RoboDK station: MiniProject.rdk

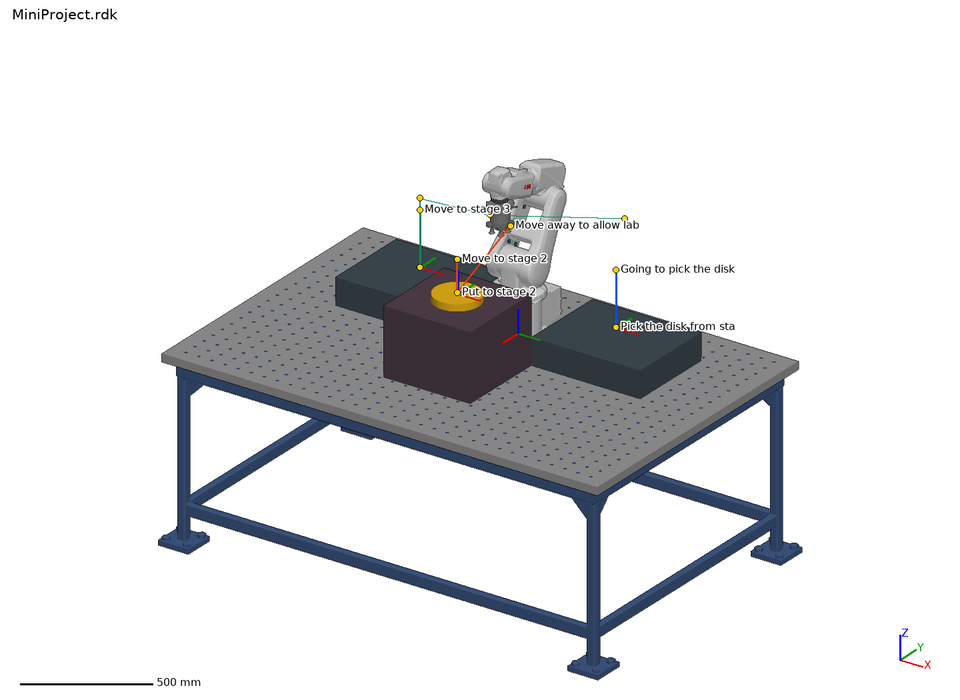
[picture v0: the station drawn from its stored meshes, robots at their saved joint values, targets as dots, program paths as lines]
Station MiniProject (saved by RoboDK 5.6.1). Poses are relative to the parent item; angles as X-Y-Z fixed-axis rotations.
  - object Table 2000x1200x800mm at (-630, -250, 0) mm, size 2020 x 1340 x 800 mm, geometry from Table-2000x1200x800mm.sld
  - object Stage 1 at (200, -200, 0) mm, size 500 x 400 x 120 mm, geometry from LINEW=0.500
  - object Stage 2 at (-200, -600, 0) mm, size 400 x 400 x 300 mm, geometry from LINEW=0.500
  - object Stage 2 at (-700, -200, 0) mm, size 500 x 400 x 120 mm, geometry from LINEW=0.500
  - frame ABB IRB 1100-4/0.58 Base at (0, 0, 0) mm, rotated rx 0 ry 0 rz -90 deg
    - robot ABB IRB 120-3/0.6: 6 axes, payload 3 kg, reach 580 mm, repeatability 0.01 mm, weight 25 kg
        modified DH rows (alpha deg, a mm, theta deg, d mm): 0, 0, 0, 290; -90, 0, -90, 0; 0, 270, 0, 0; -90, 70, 0, 302; 90, 0, 0, 0; -90, 0, 180, 72
        joint limits [-165, -110, -90, -160, -120, -400] to [165, 110, 70, 160, 120, 400]; home [0, 0, 0, 0, 0, 0]; saved at [0, -33.333, 16.582, 0, 106.741, 0]
      - tool SMC ZXP7A01-ZP20U-X1 Vacuum Gripper, TCP at (0, 0, 125) mm, size 88 x 106.8 x 127.9 mm
  - frame Frame 1 at (450, 0, 150) mm
    - target Going to pick the disk (Cartesian target) at (0, 0, 240) mm, rotated rx 180 ry 0 rz -180 deg; joints [0, 32.452, -33.546, 0, 91.094, 0] of ABB IRB 120-3/0.6
    - target Pick the disk from stage 1 (Cartesian target) at (0, 0, 0) mm, rotated rx 180 ry 0 rz -180 deg; joints [0, 47.712, -9.811, 0, 52.099, 0] of ABB IRB 120-3/0.6
  - frame Frame 2 at (0, -390, 320) mm
    - target Move to stage 2 (Cartesian target) at (0, -10, 150) mm, rotated rx 180 ry 0.01 rz 90 deg; joints [-90, 22.932, -35.32, 0, 102.378, 0] of ABB IRB 120-3/0.6
    - target Put to stage 2 (Cartesian target) at (0, -10, 10) mm, rotated rx 180 ry 0.01 rz 90 deg; joints [-90, 22.53, -7.796, 0, 75.256, 0] of ABB IRB 120-3/0.6
    - target Move away to allow label (Cartesian target) at (0, 340.58, 149.94) mm, rotated rx 180 ry 0.01 rz 90 deg; joints [-90, -49.057, 21.325, 0, 117.722, 0] of ABB IRB 120-3/0.6
    - target Pickup Again from stage 2 (Cartesian target) at (0, -10, 10) mm, rotated rx 180 ry 0.01 rz 90 deg; joints [-90, 22.53, -7.796, 0, 75.256, 0] of ABB IRB 120-3/0.6
    - target Move to up again from stage 2 (Cartesian target) at (0, -10, 150) mm, rotated rx 180 ry 0.01 rz 90 deg; joints [-90, 22.932, -35.32, 0, 102.378, 0] of ABB IRB 120-3/0.6
    - object Disk at (0, -10.01, -20) mm, rotated rx 0 ry -0.01 rz -90 deg, size 200 x 200 x 30 mm, geometry from LINEW=0.500
  - frame Frame 3 at (-450, 0, 150) mm
    - target Move to stage 3 (Cartesian target) at (0, 0, 240) mm, rotated rx -180 ry 0 rz -180 deg; joints [-180, 32.452, -33.546, 0, 91.094, 180] of ABB IRB 120-3/0.6
    - target Put on stage 2 (Cartesian target) at (0, 0, 0) mm, rotated rx -180 ry 0 rz -180 deg; joints [-180, 47.712, -9.811, 0, 52.099, 180] of ABB IRB 120-3/0.6
    - target End point 1 (Cartesian target) at (0, 0, 290) mm, rotated rx -180 ry 0 rz -180 deg; joints [-180, 34.445, -46.237, 0, 101.791, 180] of ABB IRB 120-3/0.6
    - target End Point 2 (Cartesian target) at (320, 0, 310) mm, rotated rx -180 ry 0 rz -180 deg; joints [-180, -33.964, 18.471, 0, 105.493, 180] of ABB IRB 120-3/0.6
    - target End point 3 (Cartesian target) at (939, 0, 467) mm, rotated rx 0 ry 90 rz 0 deg; joints [0, 0, 0, 0, 0, 0] of ABB IRB 120-3/0.6
  - program Replace disk 1 (1 instructions, listed below)
  - program Pick 1 (6 instructions, listed below)
  - program Place part 1 (9 instructions, listed below)
  - program Place part 2 (9 instructions, listed below)
  - program MainProgram (4 instructions, listed below)
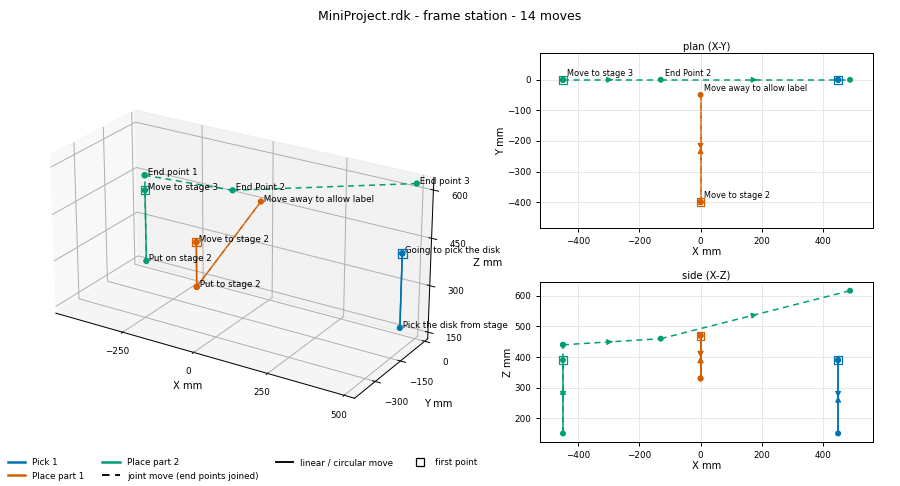
[picture p0: tool path of MiniProject.rdk in frame station, 14 of 14 moves have a stored position in this frame; points joined in program order, loops and branches not executed]

--- program Replace disk 1 (robot ABB IRB 120-3/0.6) ---
  Replace objects

--- program Pick 1 (robot ABB IRB 120-3/0.6) ---
  Set Ref.: Frame 1
  Set Tool: SMC ZXP7A01-ZP20U-X1 Vacuum Gripper
  MoveJ (Going to pick the disk)
  MoveL (Pick the disk from stage 1)
  Attach to SMC ZXP7A01-ZP20U-X1 Vacuum Gripper
  MoveL (Going to pick the disk)

--- program Place part 1 (robot ABB IRB 120-3/0.6) ---
  Set Ref.: Frame 2
  Set Tool: SMC ZXP7A01-ZP20U-X1 Vacuum Gripper
  MoveJ (Move to stage 2)
  MoveL (Put to stage 2)
  Detach from SMC ZXP7A01-ZP20U-X1 Vacuum Gripper
  MoveJ (Move away to allow label)
  MoveJ (Pickup Again from stage 2)
  Attach to SMC ZXP7A01-ZP20U-X1 Vacuum Gripper
  MoveL (Move to up again from stage 2)

--- program Place part 2 (robot ABB IRB 120-3/0.6) ---
  Set Ref.: Frame 3
  Set Tool: SMC ZXP7A01-ZP20U-X1 Vacuum Gripper
  MoveJ (Move to stage 3)
  MoveL (Put on stage 2)
  Detach from SMC ZXP7A01-ZP20U-X1 Vacuum Gripper
  MoveJ (End point) -> target End point 1
  MoveJ (End point 1)
  MoveJ (End Point 2)
  MoveJ (End point 3)

--- program MainProgram (robot ABB IRB 120-3/0.6) ---
  Call Replace disk 1
  Call Pick 1
  Call Place part 1
  Call Place part 2
